// TIA Portal project "模拟学习2" (V15.1)

(* hardware
DEVICE "S7-1200 station_1"  S7-1200 Station
   slot 0: "Rack_0"  S7-1200 Rack  Rack  V1.0
   slot 1: "PLC_1"  CPU 1212C DC/DC/DC  6ES7 212-1AE40-0XB0  V4.2
*)

// ===== PLC "PLC_1"  CPU 1212C DC/DC/DC =====

VAR_GLOBAL   // PLC tag table "默认变量表"
   ""启动"" AT %I0.0 : Bool;
   ""关闭"" AT %I0.1 : Bool;
   ""启动1"" AT %I0.2 : Bool;
   ""关闭1"" AT %I0.3 : Bool;
END_VAR